// TIA Portal V20 export
TYPE "typeCmInterfaceBrakeTest"
// stored: Access Published, Namespace Unit1.Em4
   STRUCT
      compensator : "LER_typeBrakeTestEmInterface";
      feedingRoll { S7_SetPoint := 'True'} : "LER_typeBrakeTestEmInterface";
      cutter : "LER_typeBrakeTestEmInterface";
      positionMoving { S7_SetPoint := 'True'} : "LER_typeBrakeTestEmInterface";
   END_STRUCT;
END_TYPE
